{attribute 'qualified_only'}
VAR_GLOBAL
    flag        : BOOL;             // Flag for the system
    counter     : ULINT;
    cycleTime   : LREAL := 0.001;   // Time between PLC cycles
END_VAR

VAR_GLOBAL
    otherSection : BOOL;
END_VAR

VAR_GLOBAL CONSTANT
    MY_CONST    : INT := 420;
END_VAR

VAR_GLOBAL PERSISTENT
    runtime_sec : UDINT;
END_VAR

(* stored: Version 1.1.0.1, ProductVersion 3.1.4024.11
   GVL AutoGVL: Id {3c0591f8-7ec2-40bd-a6ee-66aa6ec345bd} *)
